// SIMATIC S7-200 project (STEP 7-Micro/WIN), CPU 226 REL 02.00

ORGANIZATION_BLOCK 程序块:OB1
TITLE=MAIN:OB1
BEGIN
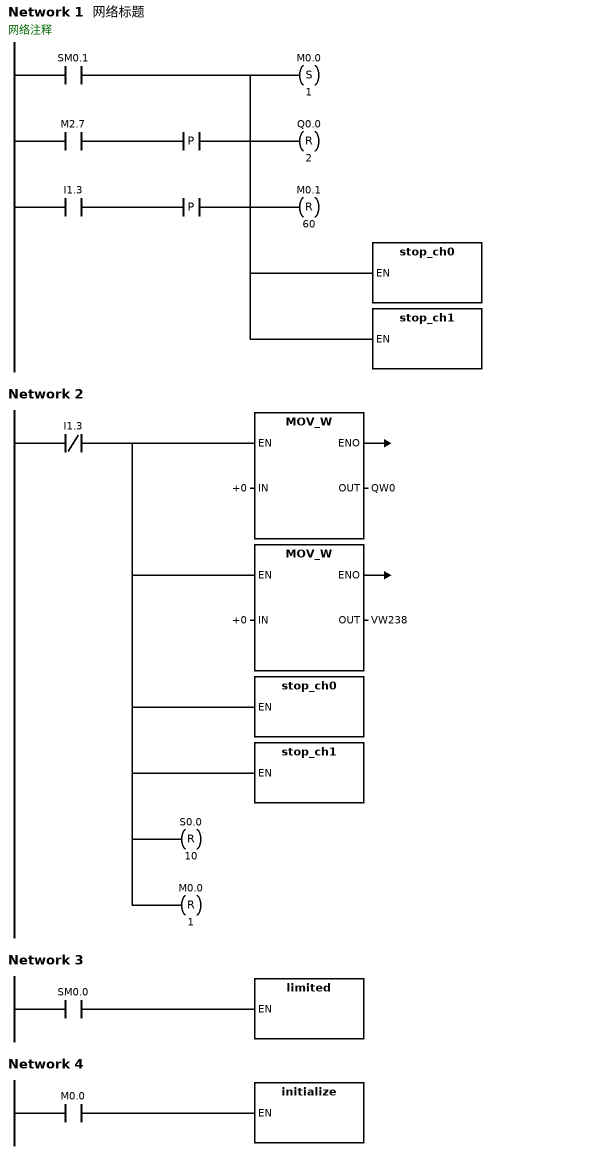
Network 1 // 网络标题
// 网络注释
LD     SM0.1
LD     M2.7
EU
OLD
LD     I1.3
EU
OLD
S      M0.0, 1
R      Q0.0, 2
R      M0.1, 60
CALL   stop_ch0:SBR6
CALL   stop_ch1:SBR8
Network 2
LDN    I1.3
MOVW   +0, QW0
MOVW   +0, VW238
CALL   stop_ch0:SBR6
CALL   stop_ch1:SBR8
R      S0.0, 10
R      M0.0, 1
Network 3
LD     SM0.0
CALL   limited:SBR1
Network 4
LD     M0.0
CALL   initialize:SBR0
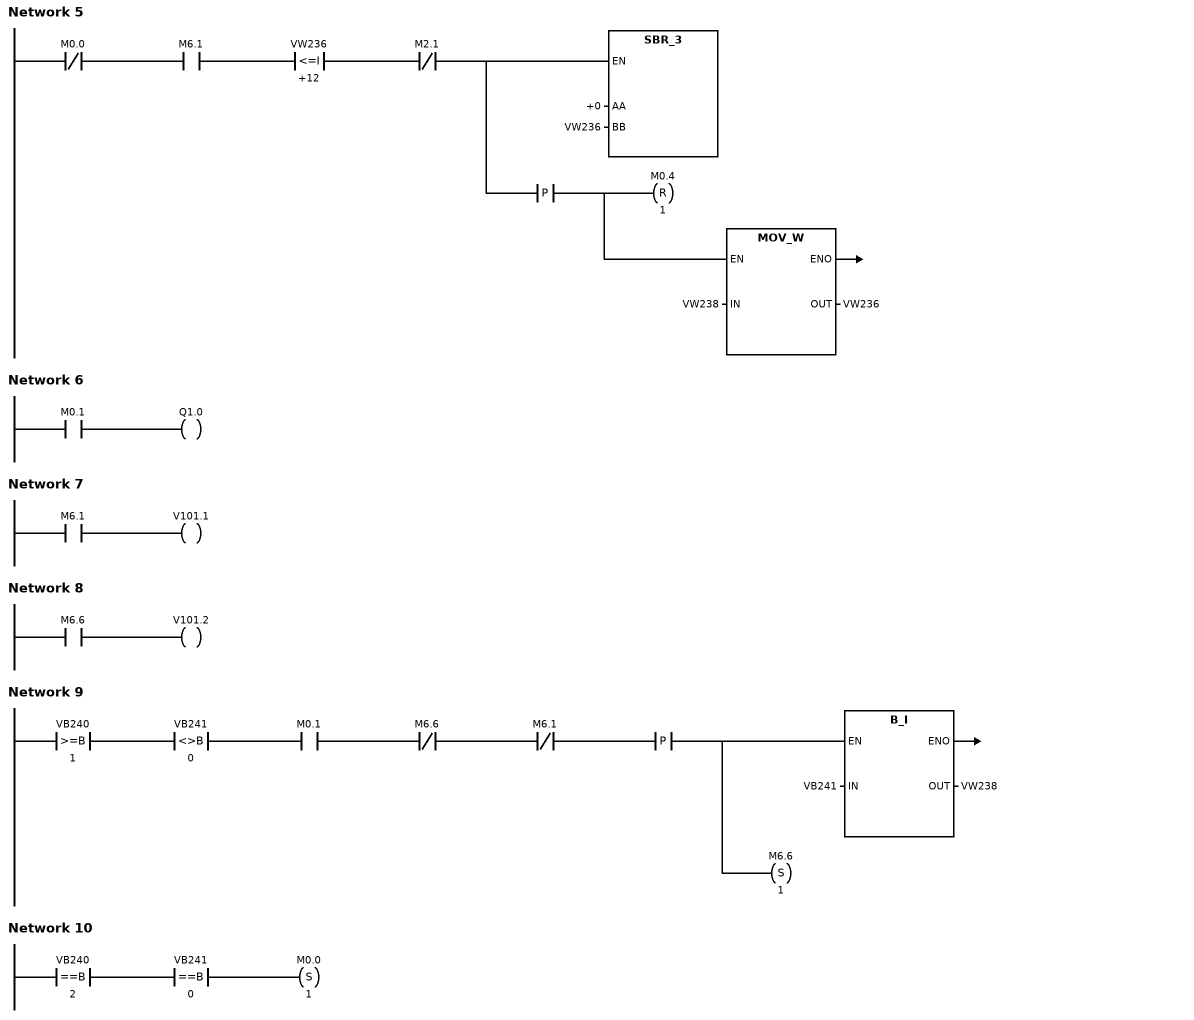
Network 5
LDN    M0.0
A      M6.1
AW<=   VW236, +12
AN     M2.1
CALL   SBR_3:SBR3, +0, VW236
EU
R      M0.4, 1
MOVW   VW238, VW236
Network 6
LD     M0.1
=      Q1.0
Network 7
LD     M6.1
=      V101.1
Network 8
LD     M6.6
=      V101.2
Network 9
LDB>=  VB240, 1
AB<>   VB241, 0
A      M0.1
AN     M6.6
AN     M6.1
EU
BTI    VB241, VW238
S      M6.6, 1
Network 10
LDB=   VB240, 2
AB=    VB241, 0
S      M0.0, 1
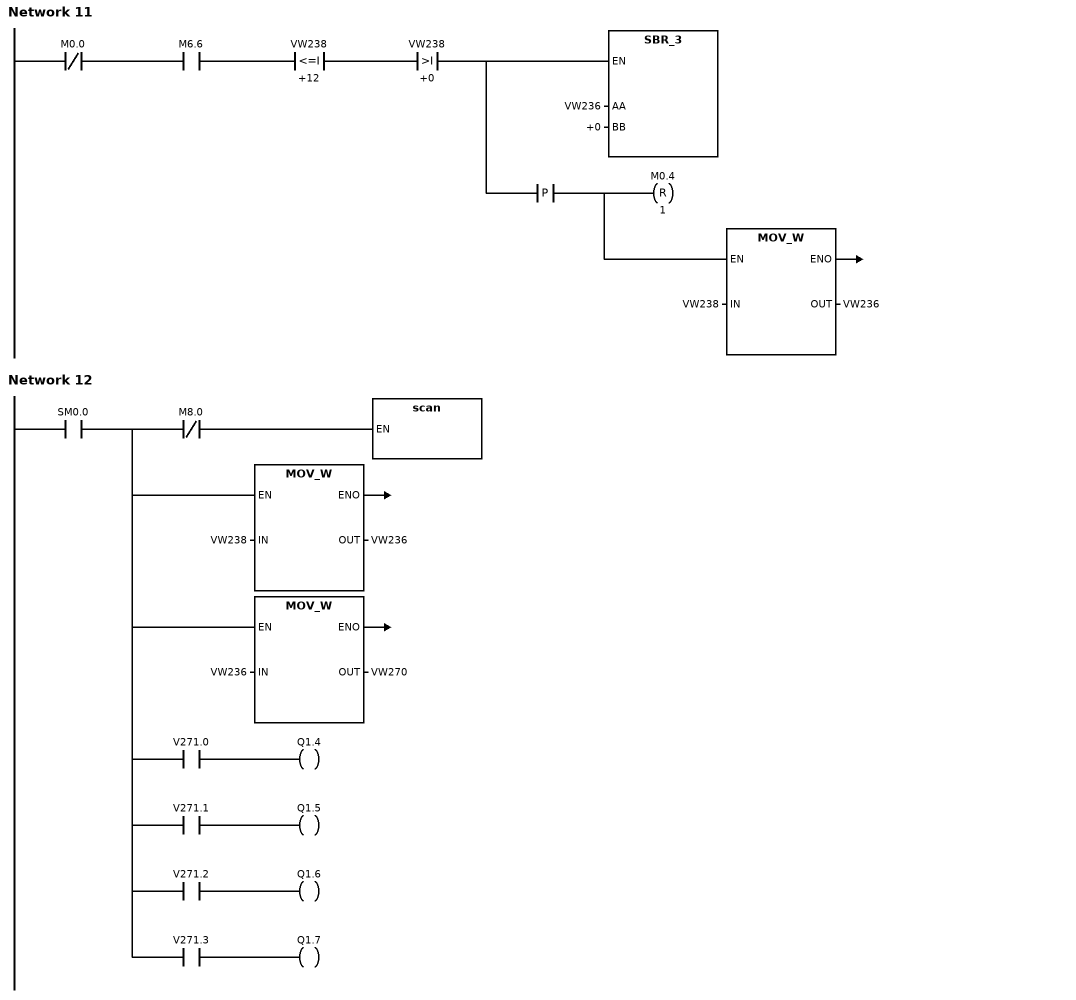
Network 11
LDN    M0.0
A      M6.6
AW<=   VW238, +12
AW>    VW238, +0
CALL   SBR_3:SBR3, VW236, +0
EU
R      M0.4, 1
MOVW   VW238, VW236
Network 12
LD     SM0.0
LPS
AN     M8.0
CALL   scan:SBR4
LRD
MOVW   VW238, VW236
LRD
MOVW   VW236, VW270
LRD
A      V271.0
=      Q1.4
LRD
A      V271.1
=      Q1.5
LRD
A      V271.2
=      Q1.6
LPP
A      V271.3
=      Q1.7
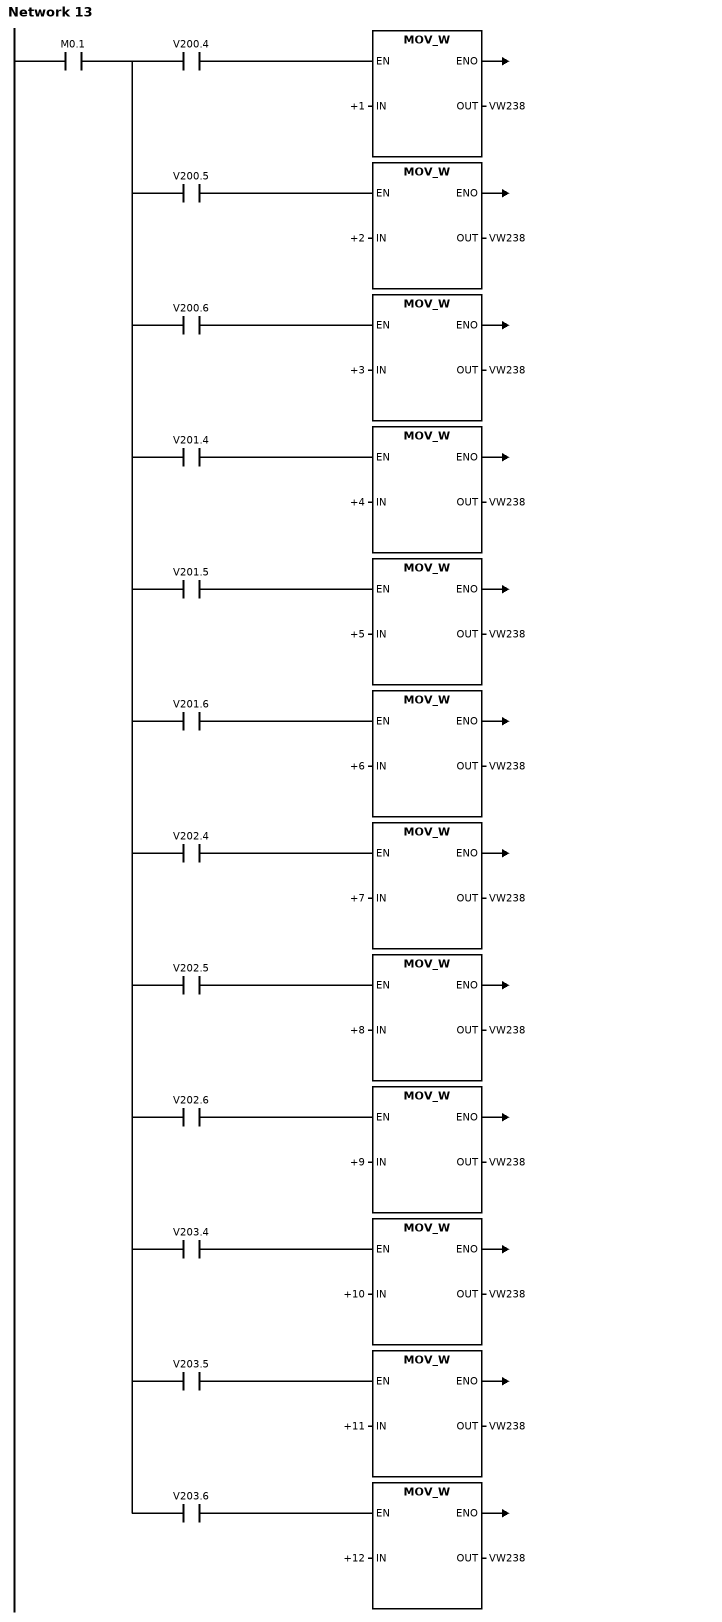
Network 13
LD     M0.1
LPS
A      V200.4
MOVW   +1, VW238
LRD
A      V200.5
MOVW   +2, VW238
LRD
A      V200.6
MOVW   +3, VW238
LRD
A      V201.4
MOVW   +4, VW238
LRD
A      V201.5
MOVW   +5, VW238
LRD
A      V201.6
MOVW   +6, VW238
LRD
A      V202.4
MOVW   +7, VW238
LRD
A      V202.5
MOVW   +8, VW238
LRD
A      V202.6
MOVW   +9, VW238
LRD
A      V203.4
MOVW   +10, VW238
LRD
A      V203.5
MOVW   +11, VW238
LPP
A      V203.6
MOVW   +12, VW238
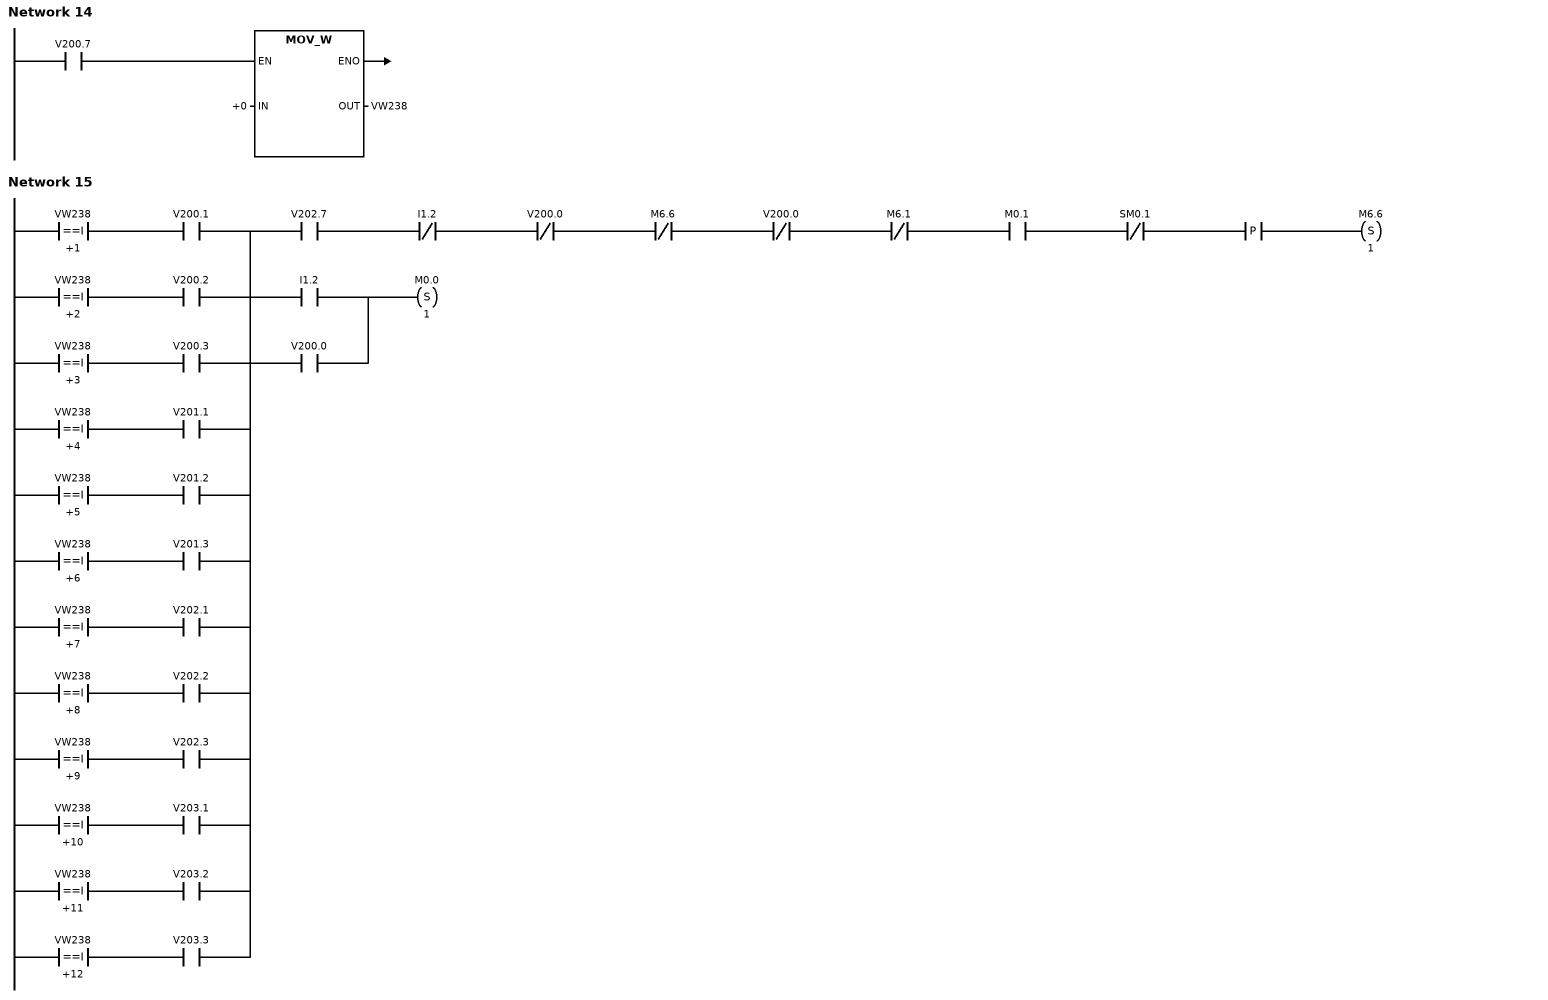
Network 14
LD     V200.7
MOVW   +0, VW238
Network 15
LDW=   VW238, +1
A      V200.1
LDW=   VW238, +2
A      V200.2
OLD
LDW=   VW238, +3
A      V200.3
OLD
LDW=   VW238, +4
A      V201.1
OLD
LDW=   VW238, +5
A      V201.2
OLD
LDW=   VW238, +6
A      V201.3
OLD
LDW=   VW238, +7
A      V202.1
OLD
LDW=   VW238, +8
A      V202.2
OLD
LDW=   VW238, +9
A      V202.3
OLD
LDW=   VW238, +10
A      V203.1
OLD
LDW=   VW238, +11
A      V203.2
OLD
LDW=   VW238, +12
A      V203.3
OLD
LPS
A      V202.7
AN     I1.2
AN     V200.0
AN     M6.6
AN     V200.0
AN     M6.1
A      M0.1
AN     SM0.1
EU
S      M6.6, 1
LPP
LD     I1.2
O      V200.0
ALD
S      M0.0, 1
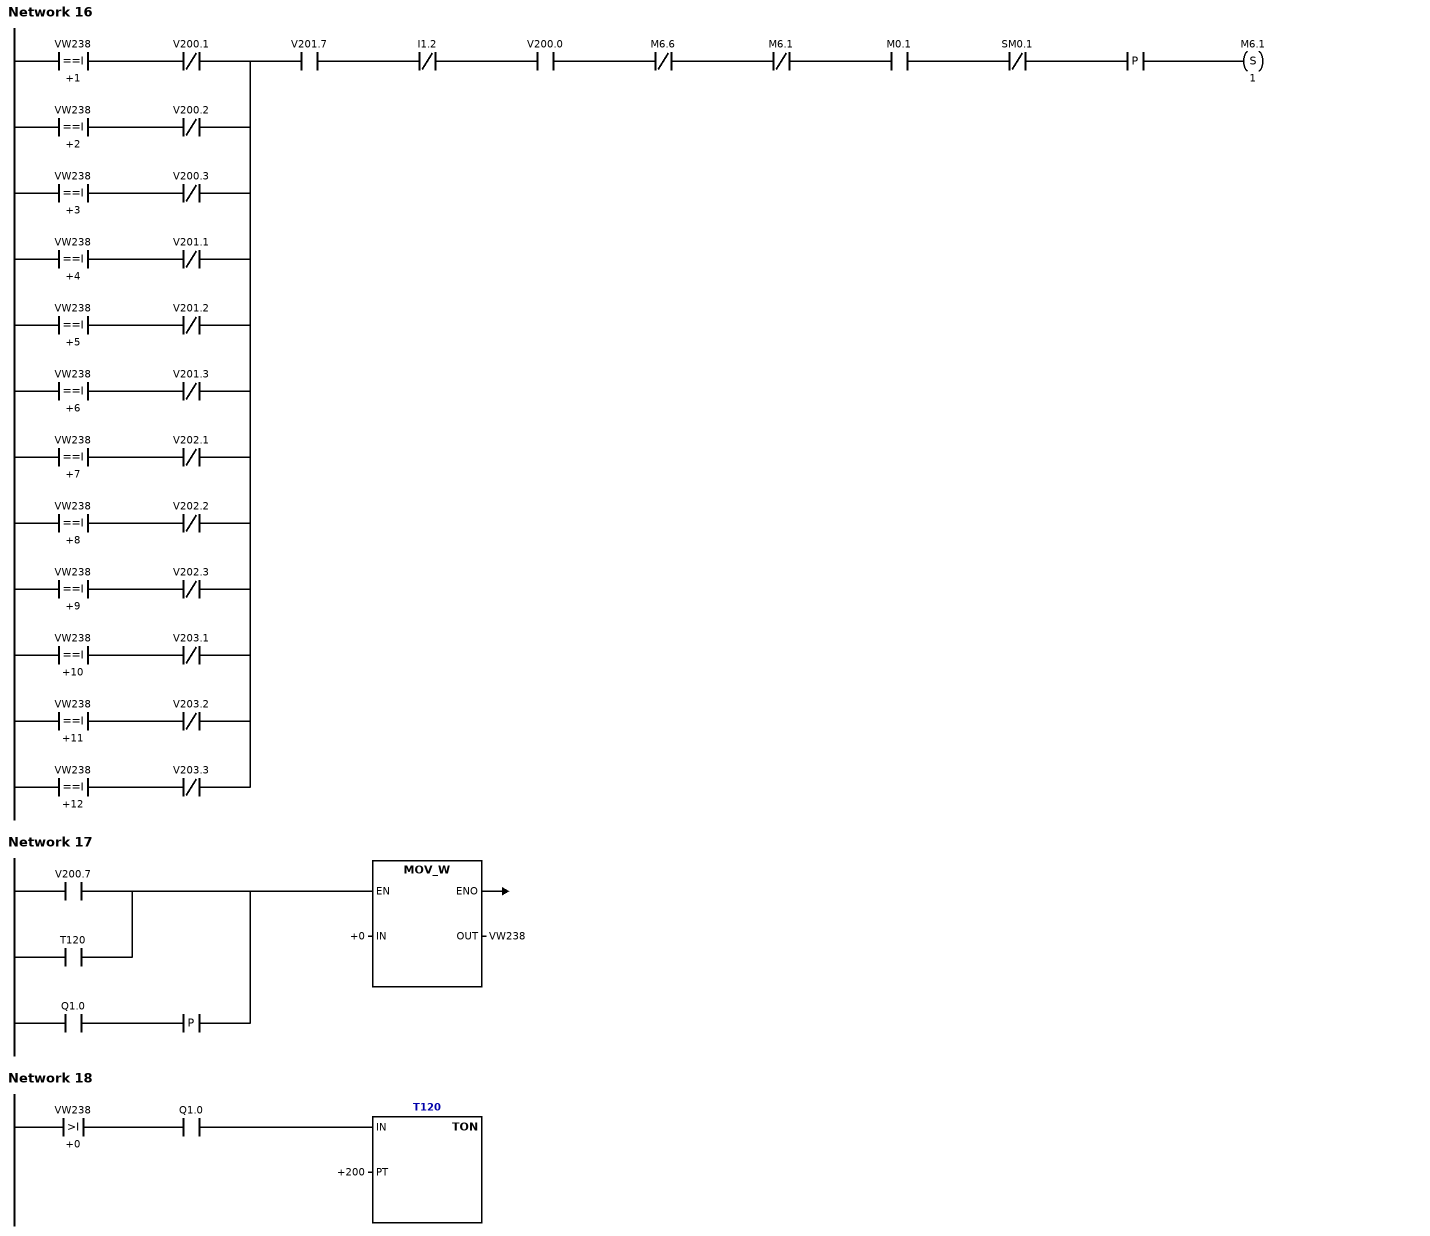
Network 16
LDW=   VW238, +1
AN     V200.1
LDW=   VW238, +2
AN     V200.2
OLD
LDW=   VW238, +3
AN     V200.3
OLD
LDW=   VW238, +4
AN     V201.1
OLD
LDW=   VW238, +5
AN     V201.2
OLD
LDW=   VW238, +6
AN     V201.3
OLD
LDW=   VW238, +7
AN     V202.1
OLD
LDW=   VW238, +8
AN     V202.2
OLD
LDW=   VW238, +9
AN     V202.3
OLD
LDW=   VW238, +10
AN     V203.1
OLD
LDW=   VW238, +11
AN     V203.2
OLD
LDW=   VW238, +12
AN     V203.3
OLD
A      V201.7
AN     I1.2
A      V200.0
AN     M6.6
AN     M6.1
A      M0.1
AN     SM0.1
EU
S      M6.1, 1
Network 17
LD     V200.7
O      T120
LD     Q1.0
EU
OLD
MOVW   +0, VW238
Network 18
LDW>   VW238, +0
A      Q1.0
TON    T120, +200
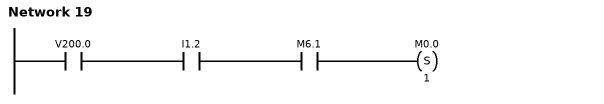
Network 19
LD     V200.0
A      I1.2
A      M6.1
S      M0.0, 1
END_ORGANIZATION_BLOCK

SUBROUTINE_BLOCK initialize:SBR0
TITLE=初始化
BEGIN
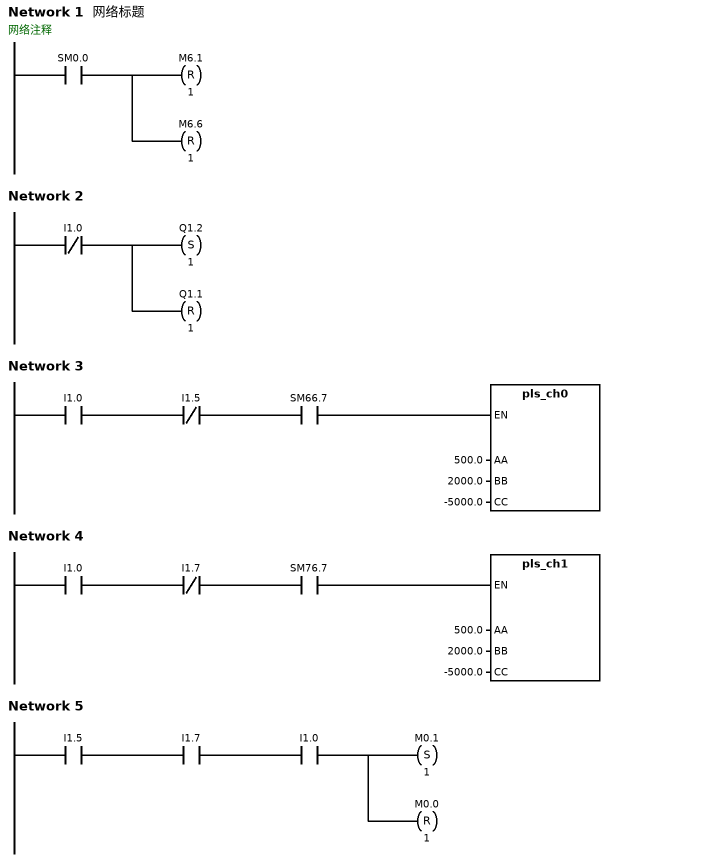
Network 1 // 网络标题
// 网络注释
LD     SM0.0
R      M6.1, 1
R      M6.6, 1
Network 2
LDN    I1.0
S      Q1.2, 1
R      Q1.1, 1
Network 3
LD     I1.0
AN     I1.5
A      SM66.7
CALL   pls_ch0:SBR5, 500.0, 2000.0, -5000.0
Network 4
LD     I1.0
AN     I1.7
A      SM76.7
CALL   pls_ch1:SBR7, 500.0, 2000.0, -5000.0
Network 5
LD     I1.5
A      I1.7
A      I1.0
S      M0.1, 1
R      M0.0, 1
END_SUBROUTINE_BLOCK

SUBROUTINE_BLOCK limited:SBR1
TITLE=限位操作
BEGIN
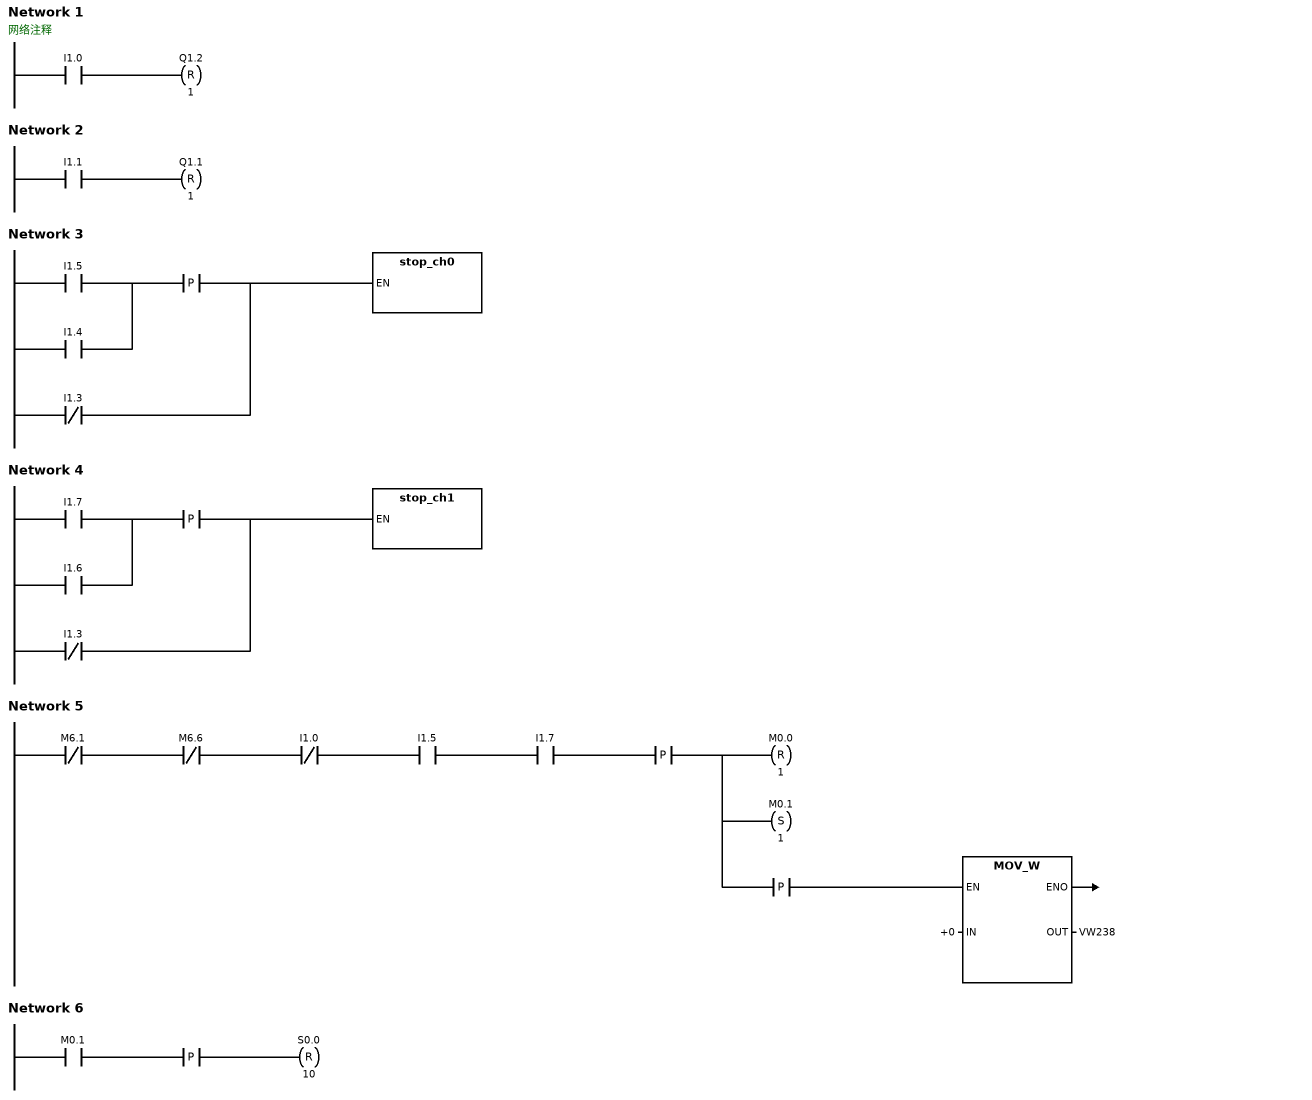
Network 1
// 网络注释
LD     I1.0
R      Q1.2, 1
Network 2
LD     I1.1
R      Q1.1, 1
Network 3
LD     I1.5
O      I1.4
EU
ON     I1.3
CALL   stop_ch0:SBR6
Network 4
LD     I1.7
O      I1.6
EU
ON     I1.3
CALL   stop_ch1:SBR8
Network 5
LDN    M6.1
AN     M6.6
AN     I1.0
A      I1.5
A      I1.7
EU
R      M0.0, 1
S      M0.1, 1
EU
MOVW   +0, VW238
Network 6
LD     M0.1
EU
R      S0.0, 10
END_SUBROUTINE_BLOCK

SUBROUTINE_BLOCK calculator:SBR2
TITLE=坐标值计算
VAR_INPUT
DEPOT:WORD;	// LW0 仓库号
END_VAR
VAR_IN_OUT
OUT_X:REAL;	// LD2 仓库X坐标
OUT_Y:REAL;	// LD6 仓库Y坐标
END_VAR
BEGIN
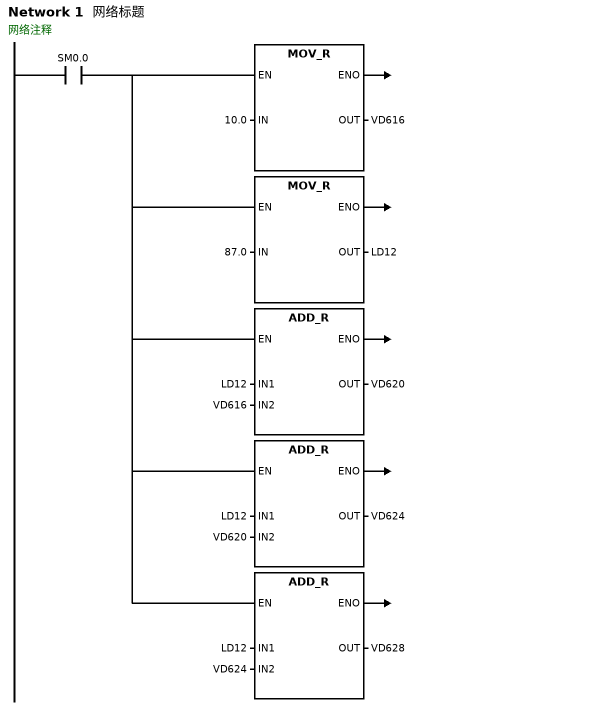
Network 1 // 网络标题
// 网络注释
LD     SM0.0
MOVR   10.0, VD616
MOVR   87.0, LD12
MOVR   LD12, VD620
+R     VD616, VD620
MOVR   LD12, VD624
+R     VD620, VD624
MOVR   LD12, VD628
+R     VD624, VD628
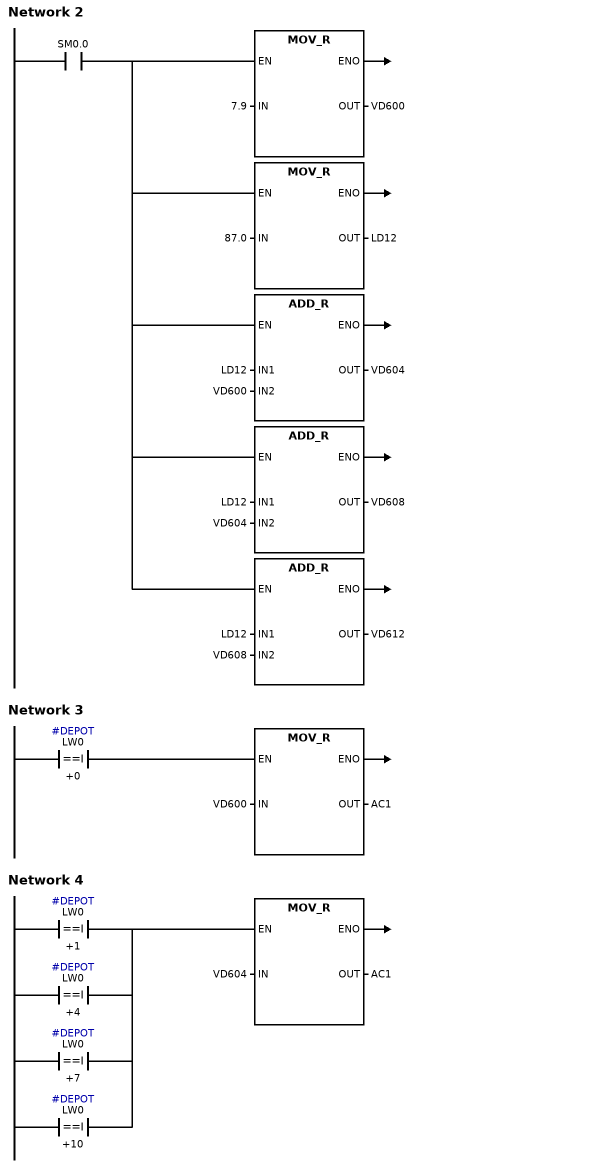
Network 2
LD     SM0.0
MOVR   7.9, VD600
MOVR   87.0, LD12
MOVR   LD12, VD604
+R     VD600, VD604
MOVR   LD12, VD608
+R     VD604, VD608
MOVR   LD12, VD612
+R     VD608, VD612
Network 3
LDW=   #DEPOT:LW0, +0
MOVR   VD600, AC1
Network 4
LDW=   #DEPOT:LW0, +1
OW=    #DEPOT:LW0, +4
OW=    #DEPOT:LW0, +7
OW=    #DEPOT:LW0, +10
MOVR   VD604, AC1
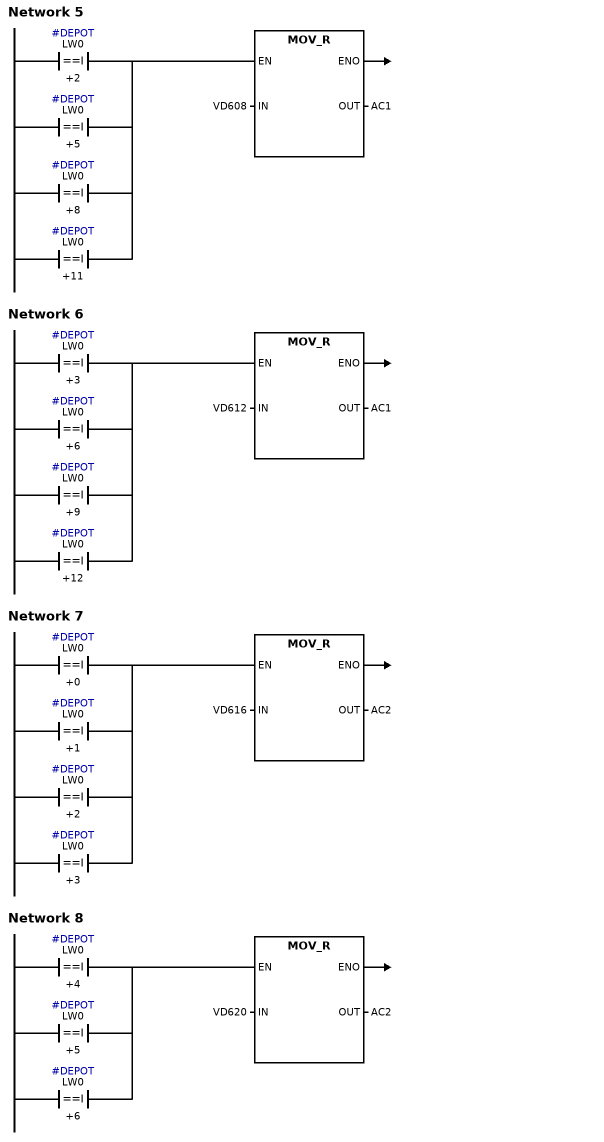
Network 5
LDW=   #DEPOT:LW0, +2
OW=    #DEPOT:LW0, +5
OW=    #DEPOT:LW0, +8
OW=    #DEPOT:LW0, +11
MOVR   VD608, AC1
Network 6
LDW=   #DEPOT:LW0, +3
OW=    #DEPOT:LW0, +6
OW=    #DEPOT:LW0, +9
OW=    #DEPOT:LW0, +12
MOVR   VD612, AC1
Network 7
LDW=   #DEPOT:LW0, +0
OW=    #DEPOT:LW0, +1
OW=    #DEPOT:LW0, +2
OW=    #DEPOT:LW0, +3
MOVR   VD616, AC2
Network 8
LDW=   #DEPOT:LW0, +4
OW=    #DEPOT:LW0, +5
OW=    #DEPOT:LW0, +6
MOVR   VD620, AC2
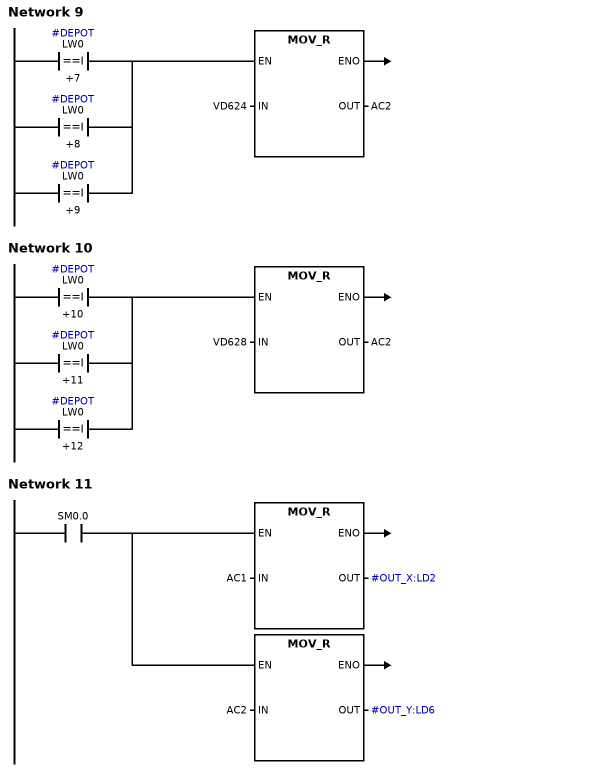
Network 9
LDW=   #DEPOT:LW0, +7
OW=    #DEPOT:LW0, +8
OW=    #DEPOT:LW0, +9
MOVR   VD624, AC2
Network 10
LDW=   #DEPOT:LW0, +10
OW=    #DEPOT:LW0, +11
OW=    #DEPOT:LW0, +12
MOVR   VD628, AC2
Network 11
LD     SM0.0
MOVR   AC1, #OUT_X:LD2
MOVR   AC2, #OUT_Y:LD6
END_SUBROUTINE_BLOCK

SUBROUTINE_BLOCK SBR_3:SBR3
TITLE=子程序4  convey:SBR3 //入库/出库操作
VAR_INPUT
AA:INT;	// LW0 
BB:WORD;	// LW2 
END_VAR
BEGIN
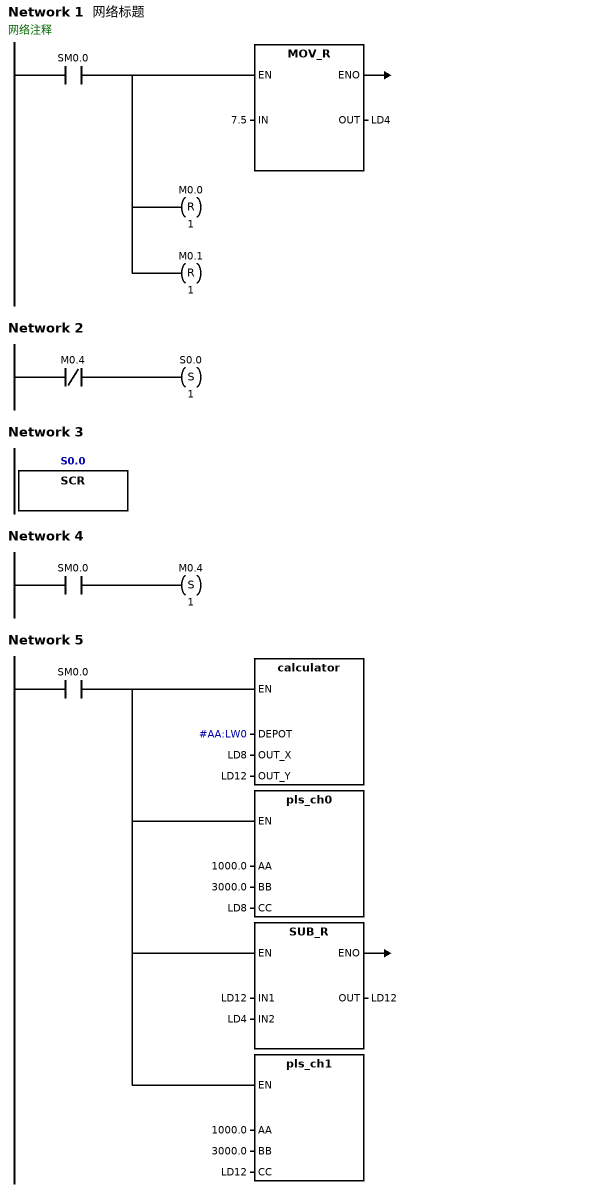
Network 1 // 网络标题
// 网络注释
LD     SM0.0
MOVR   7.5, LD4
R      M0.0, 1
R      M0.1, 1
Network 2
LDN    M0.4
S      S0.0, 1
Network 3
LSCR   S0.0
Network 4
LD     SM0.0
S      M0.4, 1
Network 5
LD     SM0.0
CALL   calculator:SBR2, #AA:LW0, LD8, LD12
CALL   pls_ch0:SBR5, 1000.0, 3000.0, LD8
-R     LD4, LD12
CALL   pls_ch1:SBR7, 1000.0, 3000.0, LD12
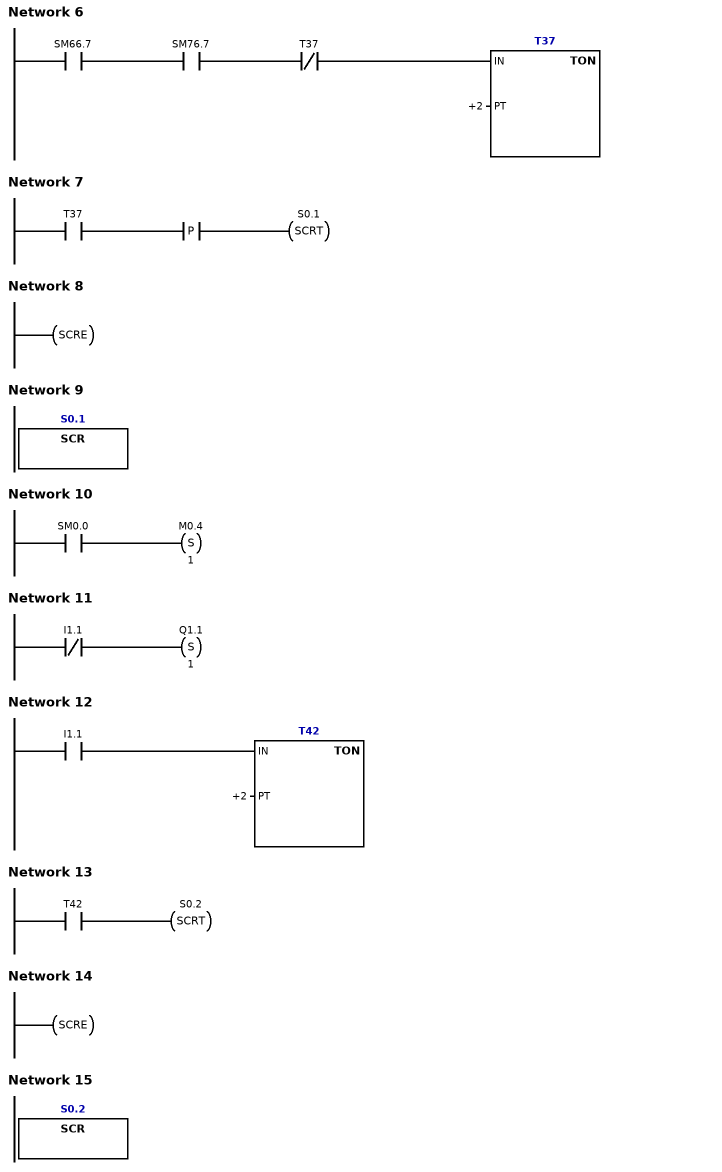
Network 6
LD     SM66.7
A      SM76.7
AN     T37
TON    T37, +2
Network 7
LD     T37
EU
SCRT   S0.1
Network 8
SCRE
Network 9
LSCR   S0.1
Network 10
LD     SM0.0
S      M0.4, 1
Network 11
LDN    I1.1
S      Q1.1, 1
Network 12
LD     I1.1
TON    T42, +2
Network 13
LD     T42
SCRT   S0.2
Network 14
SCRE
Network 15
LSCR   S0.2
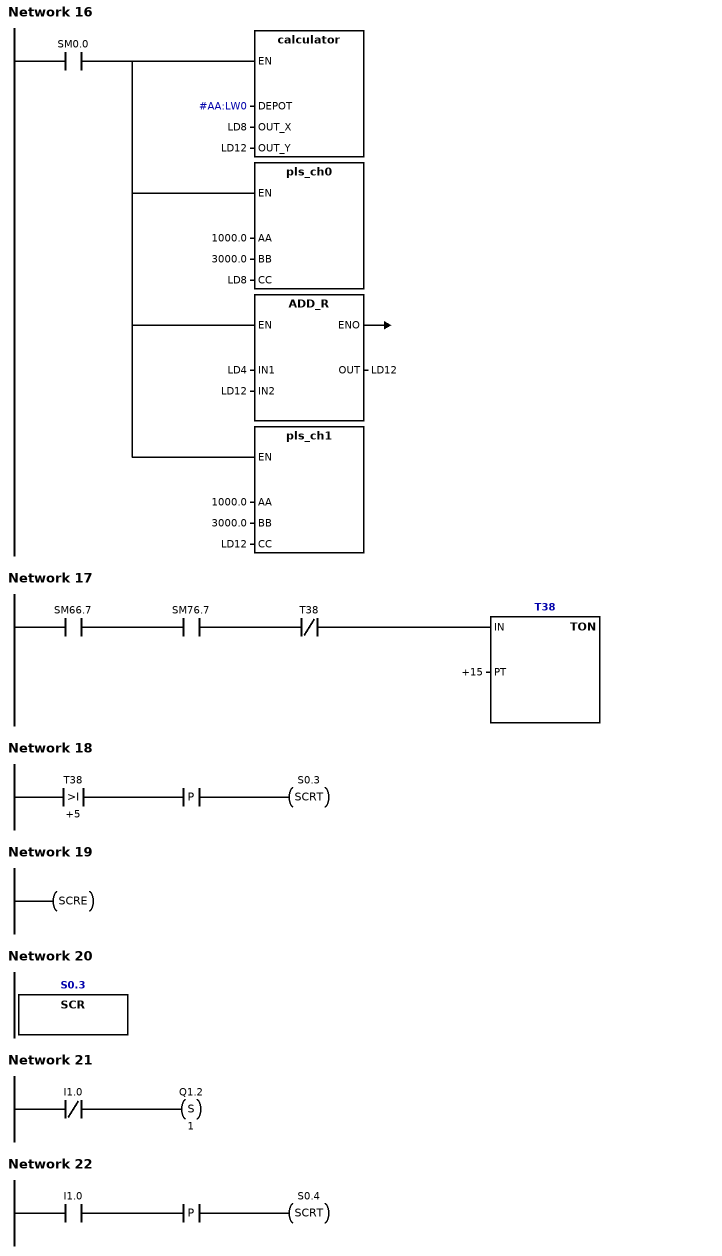
Network 16
LD     SM0.0
CALL   calculator:SBR2, #AA:LW0, LD8, LD12
CALL   pls_ch0:SBR5, 1000.0, 3000.0, LD8
+R     LD4, LD12
CALL   pls_ch1:SBR7, 1000.0, 3000.0, LD12
Network 17
LD     SM66.7
A      SM76.7
AN     T38
TON    T38, +15
Network 18
LDW>   T38, +5
EU
SCRT   S0.3
Network 19
SCRE
Network 20
LSCR   S0.3
Network 21
LDN    I1.0
S      Q1.2, 1
Network 22
LD     I1.0
EU
SCRT   S0.4
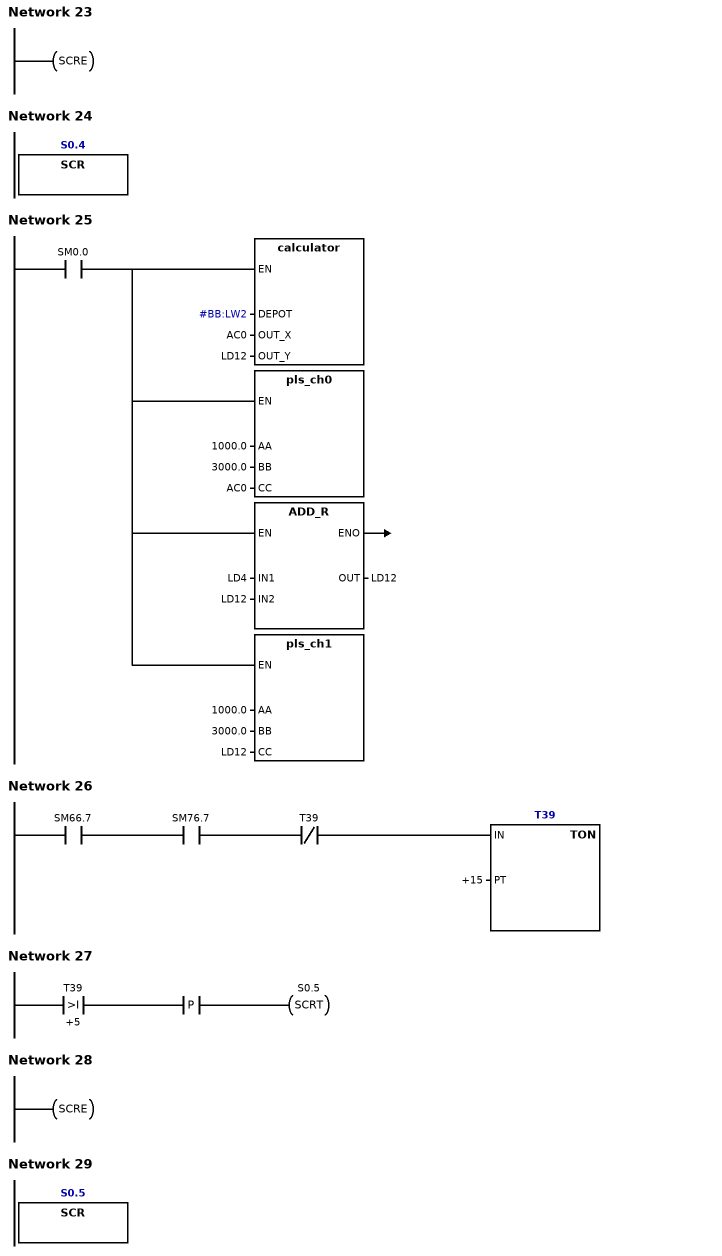
Network 23
SCRE
Network 24
LSCR   S0.4
Network 25
LD     SM0.0
CALL   calculator:SBR2, #BB:LW2, AC0, LD12
CALL   pls_ch0:SBR5, 1000.0, 3000.0, AC0
+R     LD4, LD12
CALL   pls_ch1:SBR7, 1000.0, 3000.0, LD12
Network 26
LD     SM66.7
A      SM76.7
AN     T39
TON    T39, +15
Network 27
LDW>   T39, +5
EU
SCRT   S0.5
Network 28
SCRE
Network 29
LSCR   S0.5
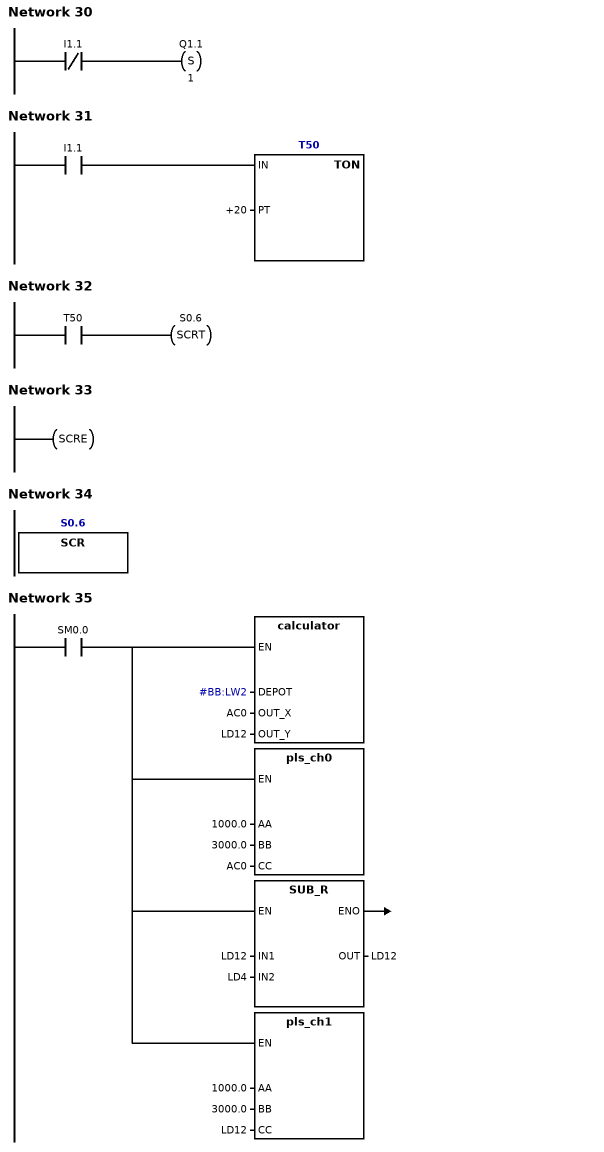
Network 30
LDN    I1.1
S      Q1.1, 1
Network 31
LD     I1.1
TON    T50, +20
Network 32
LD     T50
SCRT   S0.6
Network 33
SCRE
Network 34
LSCR   S0.6
Network 35
LD     SM0.0
CALL   calculator:SBR2, #BB:LW2, AC0, LD12
CALL   pls_ch0:SBR5, 1000.0, 3000.0, AC0
-R     LD4, LD12
CALL   pls_ch1:SBR7, 1000.0, 3000.0, LD12
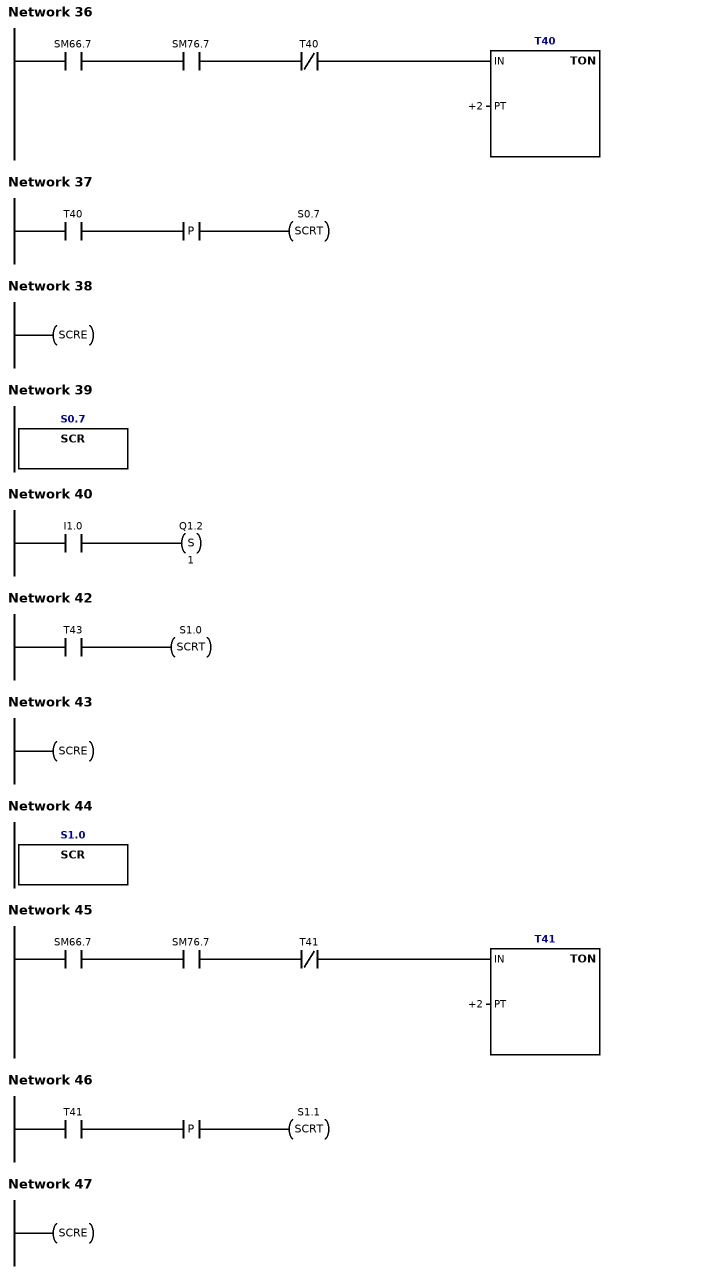
Network 36
LD     SM66.7
A      SM76.7
AN     T40
TON    T40, +2
Network 37
LD     T40
EU
SCRT   S0.7
Network 38
SCRE
Network 39
LSCR   S0.7
Network 40
LD     I1.0
S      Q1.2, 1
Network 41
LDN    I1.0
TON    T43, +2
LDN    I1.0
TON    T43, +2
Network 42
LD     T43
SCRT   S1.0
Network 43
SCRE
Network 44
LSCR   S1.0
Network 45
LD     SM66.7
A      SM76.7
AN     T41
TON    T41, +2
Network 46
LD     T41
EU
SCRT   S1.1
Network 47
SCRE
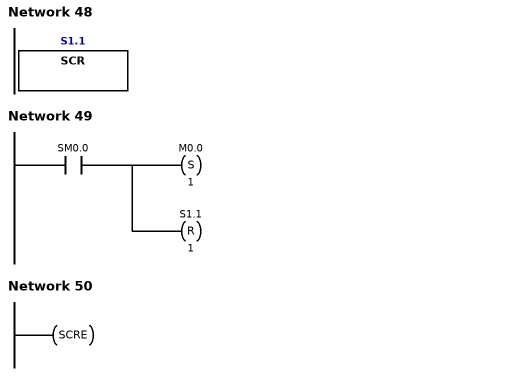
Network 48
LSCR   S1.1
Network 49
LD     SM0.0
S      M0.0, 1
R      S1.1, 1
Network 50
SCRE
END_SUBROUTINE_BLOCK

SUBROUTINE_BLOCK scan:SBR4
TITLE=子程序5//键盘扫描程序
BEGIN
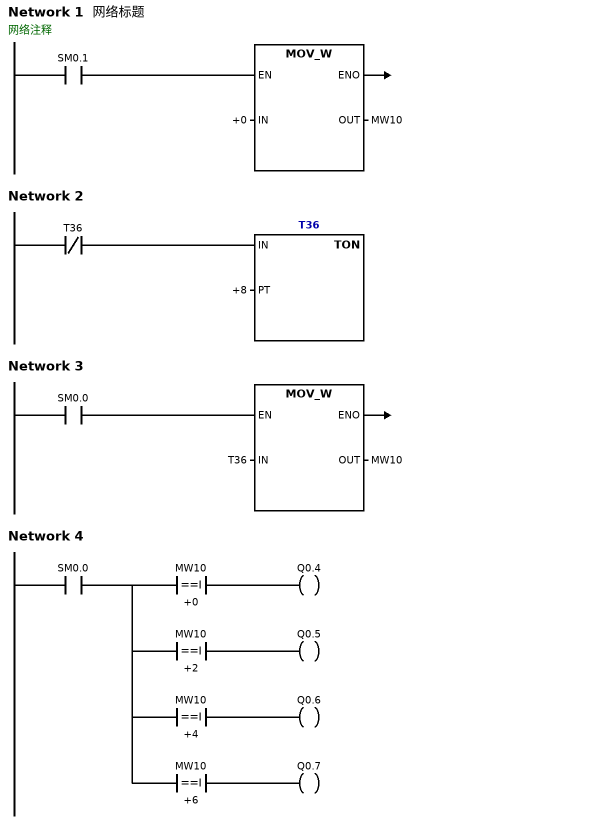
Network 1 // 网络标题
// 网络注释
LD     SM0.1
MOVW   +0, MW10
Network 2
LDN    T36
TON    T36, +8
Network 3
LD     SM0.0
MOVW   T36, MW10
Network 4
LD     SM0.0
LPS
AW=    MW10, +0
=      Q0.4
LRD
AW=    MW10, +2
=      Q0.5
LRD
AW=    MW10, +4
=      Q0.6
LPP
AW=    MW10, +6
=      Q0.7
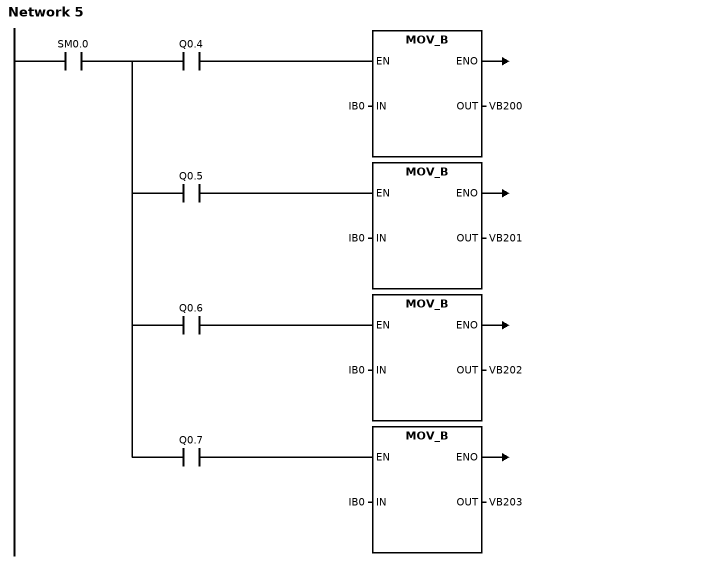
Network 5
LD     SM0.0
LPS
A      Q0.4
MOVB   IB0, VB200
LRD
A      Q0.5
MOVB   IB0, VB201
LRD
A      Q0.6
MOVB   IB0, VB202
LPP
A      Q0.7
MOVB   IB0, VB203
END_SUBROUTINE_BLOCK

SUBROUTINE_BLOCK pls_ch0:SBR5
TITLE=子程序6    //脉冲发生器1的控制程序
VAR_INPUT
AA:REAL;	// LD0 
BB:REAL;	// LD4 
CC:REAL;	// LD8 
END_VAR
BEGIN
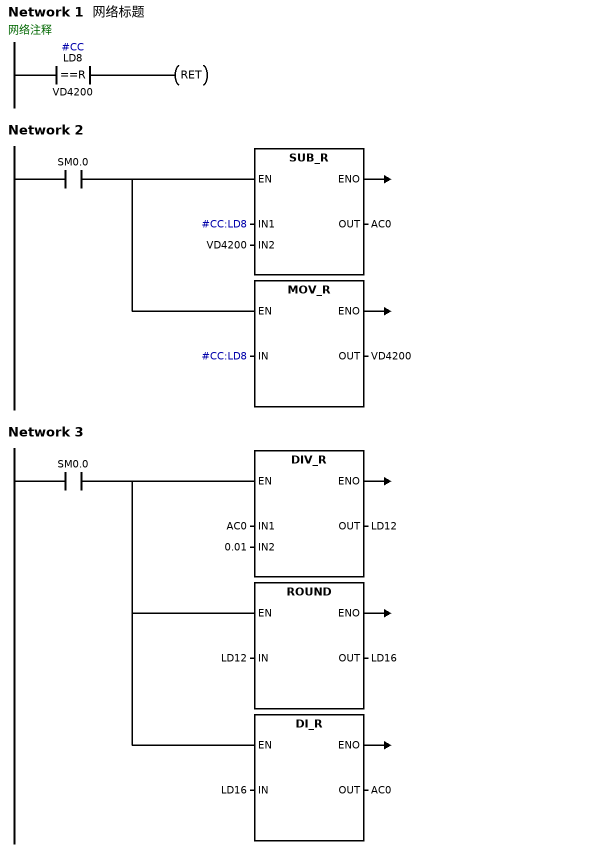
Network 1 // 网络标题
// 网络注释
LDR=   #CC:LD8, VD4200
CRET
Network 2
LD     SM0.0
MOVR   #CC:LD8, AC0
-R     VD4200, AC0
MOVR   #CC:LD8, VD4200
Network 3
LD     SM0.0
MOVR   AC0, LD12
/R     0.01, LD12
ROUND  LD12, LD16
DTR    LD16, AC0
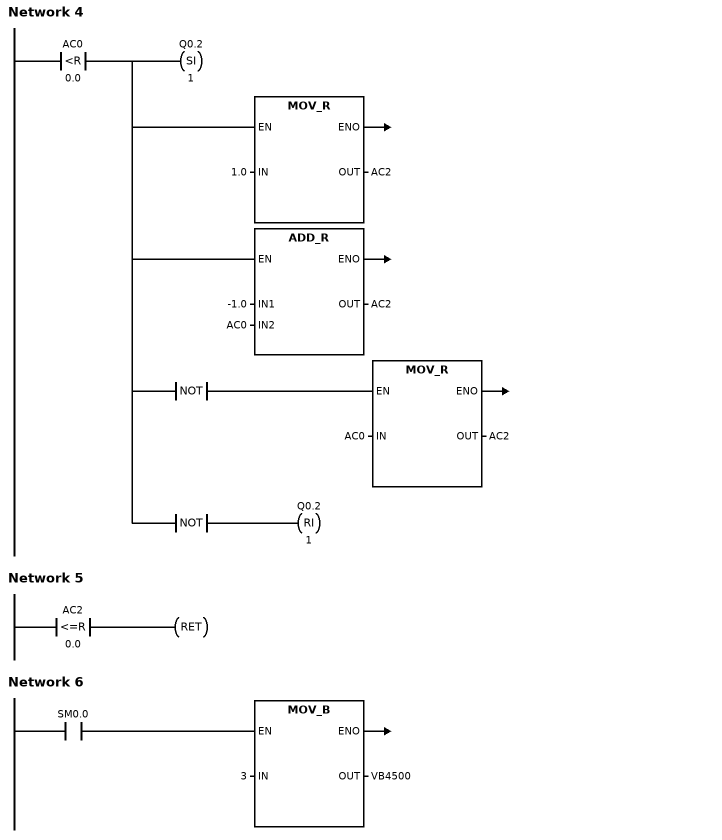
Network 4
LDR<   AC0, 0.0
LPS
SI     Q0.2, 1
MOVR   1.0, AC2
MOVR   -1.0, AC2
+R     AC0, AC2
NOT
MOVR   AC0, AC2
LPP
NOT
RI     Q0.2, 1
Network 5
LDR<=  AC2, 0.0
CRET
Network 6
LD     SM0.0
MOVB   3, VB4500
